// function block for inductive sensor with the option of debouncing + rising and falling edge detection.
FUNCTION_BLOCK FB_Component_InductiveSensor IMPLEMENTS  I_Component
VAR_INPUT
	bSignal			: BOOL;				// Raw input sensor
	tDebounce		: TIME := T#0MS;	// Debounce time
// Interface vars
	sName			: STRING[20];
	bEnable     	: BOOL;
	//eMode       	: E_ComponentMode;
END_VAR

VAR_OUTPUT
	bActive			: BOOL;
	bRising			: BOOL;
	bFalling		: BOOL;
// interface vars
	eState			: E_ComponentState;
	iErrorCode		: INT;
	sStatusText 	: STRING[50];
END_VAR

VAR
	bLastSignal		: BOOL;
	tDebTimer		: TON;
	bSignalStable	: BOOL;
END_VAR

IF bEnable AND eState = (E_ComponentState.READY OR E_ComponentState.BUSY) THEN
	IF bLastSignal <> bSignal THEN
		tDebTimer(IN := TRUE, PT := tDebounce);
		eState := E_ComponentState.BUSY;
	ELSE
		tDebTimer(IN := FALSE);
	END_IF
	
	IF tDebTimer.Q THEN
		bSignalStable 	:= bSignal;
		bLastSignal 	:= bSignal;
		eState := E_ComponentState.READY;
	END_IF
	
	bRising		:= (bSignalStable AND NOT bActive);
	bFalling	:= (NOT bSignalStable AND bActive);
	bActive 	:= bSignalStable;
ELSE
	bActive 	:= FALSE;
	bRising		:= FALSE;
	bFalling	:= FALSE;
	tDebTimer(IN := FALSE);
END_IF

METHOD Halt : BOOL
bActive 	:= FALSE;
bRising		:= FALSE;
bFalling	:= FALSE;
tDebTimer(IN := FALSE);
eState := E_ComponentState.HALTED;
END_METHOD

METHOD Start : BOOL
eState := E_ComponentState.READY;
END_METHOD

METHOD Stop : BOOL
IF eState <> E_ComponentState.BUSY THEN
	bActive 	:= FALSE;
	bRising		:= FALSE;
	bFalling	:= FALSE;
	eState := E_ComponentState.DONE;
END_IF
END_METHOD

END_FUNCTION_BLOCK

(* stored: Version 1.1.0.1, ProductVersion 3.1.4024.15
   POU FB_Component_InductiveSensor: Id {8e7ef9e5-be5c-4d5b-9caf-29f0d28584ab}, SpecialFunc None
   Method Halt: Id {f3238e3e-c657-463e-ba29-1e530a523711}
   Method Start: Id {332d80dd-0194-4918-b2f7-7e712950268d}
   Method Stop: Id {1e590e11-4492-46f6-8aed-701c371c3bb9} *)
